// TIA Portal project "plc hmi game" (V17)

(* hardware
DEVICE "HMI_1"  KTP400 Basic PN
   slot 0: "HMI_1"  KTP400 Basic PN  6AV2 123-2DB03-0AX0  15.1.0.0
   slot 1: "HMI_RT_1"  KTP400 Basic PN  6AV2 123-2DB03-0AX0  15.1.0.0
   slot 5: "HMI_1.IE_CP_1"  PROFINET Interface  15.0.1.0
      slot 1: "PROFINET Interface_1"  PROFINET Interface
         slot 1: "Port_1"  Port
DEVICE "S7-1200 station_1"  S7-1200 Station
   slot 0: "Rack_0"  S7-1200 Rack  Rack  V1.0
   slot 1: "PLC_1"  CPU 1211C DC/DC/DC  6ES7 211-1AE40-0XB0  V4.5
*)

// ===== PLC "PLC_1"  CPU 1211C DC/DC/DC =====

VAR_GLOBAL   // PLC tag table "Default tag table"
   "baloon_jump" AT %M0.2 : Bool;
   "Tag_2" AT %M1.0 : Bool;
   "baloon" AT %MW10 : Word;
   "Tag_1" AT %MW0 : Word;
   "Tag_3" AT %MD0 : Time;
   "Tag_4" AT %MW6 : Word;
   "Tag_5" AT %M0.0 : Bool;
   "Tag_6" AT %M0.3 : Bool;
   "Tag_7" AT %M0.4 : Bool;
   "Tag_8" AT %MW12 : Word;
   "Tag_9" AT %MD12 : Time;
   "Tag_10" AT %MW4 : Word;
   "Tag_11" AT %M0.6 : Bool;
   "Tag_12" AT %MW8 : Word;
   "Tag_13" AT %M0.7 : Bool;
   "Tag_14" AT %M0.1 : Bool;
   "Tag_15" AT %M2.0 : Bool;
END_VAR

// folder: System blocks/Program resources

DATA_BLOCK "IEC_Timer_0_DB"   // DB1
{ S7_Optimized_Access := 'TRUE' }
AUTHOR : Simatic
FAMILY : IEC
NAME : IEC_TMR
VERSION : 1.0
// stored: InstanceOfName IEC_TIMER
"IEC_TIMER"
BEGIN
END_DATA_BLOCK

DATA_BLOCK "IEC_Timer_0_DB_1"   // DB2
{ S7_Optimized_Access := 'TRUE' }
AUTHOR : Simatic
FAMILY : IEC
NAME : IEC_TMR
VERSION : 1.0
// stored: InstanceOfName IEC_TIMER
"IEC_TIMER"
BEGIN
END_DATA_BLOCK

DATA_BLOCK "IEC_Timer_0_DB_2"   // DB3
{ S7_Optimized_Access := 'TRUE' }
AUTHOR : Simatic
FAMILY : IEC
NAME : IEC_TMR
VERSION : 1.0
// stored: InstanceOfName IEC_TIMER
"IEC_TIMER"
BEGIN
END_DATA_BLOCK

// folder: (top level)

ORGANIZATION_BLOCK "Main"   // OB1, LAD, ProgramCycle
TITLE = "Main Program Sweep (Cycle)"
{ S7_Optimized_Access := 'TRUE' }
VERSION : 0.1
   VAR_INPUT
      Initial_Call : Bool;   // Initial call of this OB
      Remanence : Bool;   // =True, if remanent data are available
   END_VAR
BEGIN

REGION Network 1
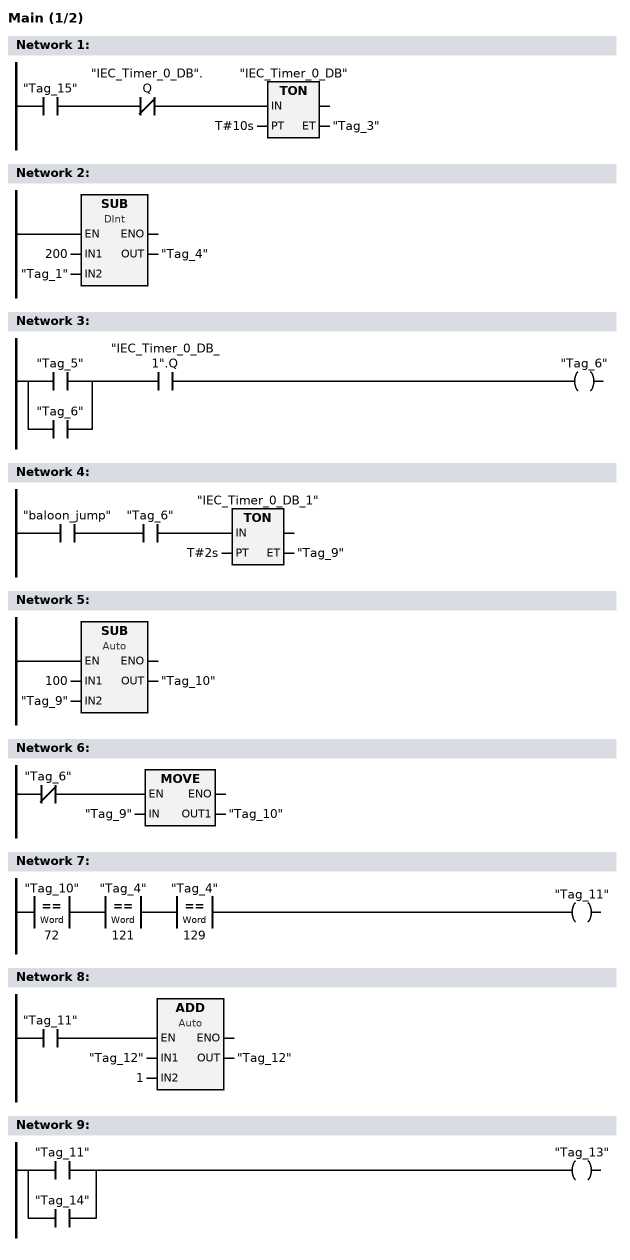
   "IEC_Timer_0_DB".TON(IN := "Tag_15" AND NOT "IEC_Timer_0_DB".Q, PT := T#10s, ET => "Tag_3");
END_REGION

REGION Network 2
   RUNG wire#powerrail
      { S7_Templates := "SrcType := DInt" } Sub(in1 := 200, in2 := "Tag_1", out => "Tag_4")
   END_RUNG
   // the same network as SCL:
   "Tag_4" := 200 - "Tag_1";
END_REGION

REGION Network 3
   RUNG wire#powerrail
      Contact( "Tag_5" )
      wire#w1
      Contact( "IEC_Timer_0_DB_1".Q )
      Coil( "Tag_6" )
   END_RUNG
   RUNG wire#powerrail
      Contact( "Tag_6" )
   END_RUNG wire#w1
   // the same network as SCL:
   "Tag_6" := ("Tag_5" OR "Tag_6") AND "IEC_Timer_0_DB_1".Q;
END_REGION

REGION Network 4
   "IEC_Timer_0_DB_1".TON(IN := "baloon_jump" AND "Tag_6", PT := T#2s, ET => "Tag_9");
END_REGION

REGION Network 5
   RUNG wire#powerrail
      Sub(in1 := 100, in2 := "Tag_9", out => "Tag_10")
   END_RUNG
   // the same network as SCL:
   "Tag_10" := 100 - "Tag_9";
END_REGION

REGION Network 6
   RUNG wire#powerrail
      I_Contact( "Tag_6" )
      Move(in := "Tag_9", out1 => "Tag_10")
   END_RUNG
   // the same network as SCL:
   IF NOT "Tag_6" THEN "Tag_10" := "Tag_9"; END_IF;
END_REGION

REGION Network 7
   RUNG wire#powerrail
      { S7_Templates := "SrcType := Word" } EQ_Contact(in1 := "Tag_10", in2 := 72)
      { S7_Templates := "SrcType := Word" } EQ_Contact(in1 := "Tag_4", in2 := 121)
      { S7_Templates := "SrcType := Word" } EQ_Contact(in1 := "Tag_4", in2 := 129)
      Coil( "Tag_11" )
   END_RUNG
   // the same network as SCL:
   "Tag_11" := ("Tag_10" = 72) AND ("Tag_4" = 121) AND ("Tag_4" = 129);
END_REGION

REGION Network 8
   RUNG wire#powerrail
      Contact( "Tag_11" )
      Add(in1 := "Tag_12", in2 := 1, out => "Tag_12")
   END_RUNG
   // the same network as SCL:
   IF "Tag_11" THEN "Tag_12" := "Tag_12" + 1; END_IF;
END_REGION

REGION Network 9
   RUNG wire#powerrail
      Contact( "Tag_11" )
      wire#w1
      Coil( "Tag_13" )
   END_RUNG
   RUNG wire#powerrail
      Contact( "Tag_14" )
   END_RUNG wire#w1
   // the same network as SCL:
   "Tag_13" := "Tag_11" OR "Tag_14";
END_REGION

REGION Network 10
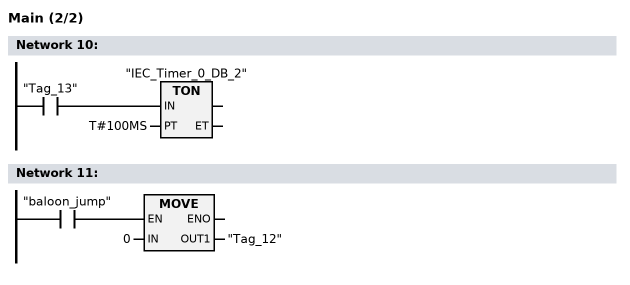
   "IEC_Timer_0_DB_2".TON(IN := "Tag_13", PT := T#100MS);
END_REGION

REGION Network 11
   RUNG wire#powerrail
      Contact( "baloon_jump" )
      Move(in := 0, out1 => "Tag_12")
   END_RUNG
   // the same network as SCL:
   IF "baloon_jump" THEN "Tag_12" := 0; END_IF;
END_REGION
END_ORGANIZATION_BLOCK

(* ===== HMI "HMI_RT_1" =====
system functions are stored by id; their names below are inferred from use
connection "Connection_1": ETHERNET, SMART_S7_1200_OMS
connection "HMI_Connection_1": ETHERNET, SMART_S7_1200_OMS

HMI tags "Default tag table"
   "Tag_5(1)" : Bool = PLC Tag_5 AT %M0.0, 1 s
   "TAG_2" : Bool = PLC Tag_14 AT %M0.1, 1 s
   "TAG_3" : Word = PLC Tag_10 AT %MW4, 1 s
   "TAG_4" : Word = PLC Tag_4 AT %MW6, 1 s
   "TAG_5" : Word = PLC Tag_12 AT %MW8, 1 s
   "TAG_6" : Bool = PLC baloon_jump AT %M0.2, 1 s

Template "Template_1" 480x272
   Button "Exit" at 388,227 size 63x44; TextOff 'Exit'; PictureOff "ExitRuntime_KTP400_Basic_PN_TR"; PictureOn "ExitRuntime_KTP400_Basic_PN_TR"
      on Release: StopRuntime(0)
   Button "Template_Button" at 268,227 size 63x44; TextOff 'Text'
   Button "Alarms" at 148,227 size 63x44; TextOff 'Alarms'; PictureOff "AlarmDisplay_KTP400_Basic_PN_TR"; PictureOn "AlarmDisplay_KTP400_Basic_PN_TR"
      on Release: function_ef3f5d25("Alarm window_Unacknowledged", -1)
   Button "Start screen" at 28,227 size 63x44; TextOff 'Start screen'; PictureOff "NavigateHome_KTP400_Basic_PN_TR"; PictureOn "NavigateHome_KTP400_Basic_PN_TR"
   SymbolicIOField "Symbolic_IO_Field_Screen" at 82,8 size 311x29; TextOff '0'; TextOn '1'; TextList "TextList_ScreenNames"
      ProcessValue <- "Tag_5(1)"
      on Change: ActivateScreenByNumber("TAG_5", 0)
   DateTimeField "HmiScreenItemData" at 395,22 size 85x22
   DateTimeField "HmiScreenItemData_1" at 395,0 size 85x22
   GraphicView "Logo" at 0,0 size 80x45; Picture "Logo of HMI_1"

screen "Screen_1" 480x272
   Button "Button_1" at 190,86 size 96x32; TextOff 'ENTER'
      on Press: ActivateScreen("Screen_2", 0)

screen "Screen_2" 480x272
   Button "Button_1" at 6,14 size 76x24; TextOff 'ENTER'
      on Click: InvertBit("TAG_6")
   Button "Button_2" at 7,39 size 76x24; TextOff 'EXIT'
      on Click: StopRuntime(0)
   GraphicView "Graphic view_1" at 0,136 size 73x29; Picture "Graphic_1"
   GraphicView "Graphic view_2" at 102,136 size 36x30; Picture "Graphic_2"
      Visibility <- "TAG_2"
      HorizontalMovement <- "TAG_3"
   IOField "I/O field_1" at 373,21 size 96x32; FormatPattern 99999
      ProcessValue <- "TAG_5"
   Ellipse "Ellipse_1" at 215,39 size 64x25
      Visibility <- "TAG_2"
      VerticalMovement <- "TAG_4"
   Button "Button_3" at 6,224 size 96x32; TextOff 'FIRE'
      on Release: ResetBit("Tag_5(1)")
      on Press: SetBit("Tag_5(1)")
   Button "Button_4" at 388,235 size 84x24; TextOff 'BACK'
      on Press: function_efd93a16()
   GraphicView "Graphic view_3" at 233,137 size 36x30; Picture "Graphic_3"
      Visibility <- "TAG_2"
*)